{attribute 'qualified_only'}
VAR_GLOBAL
	DigIn AT %I*:ARRAY[1..16]	OF	BOOL;
	DigOut1 AT %Q*:ARRAY[1..4]	OF	BOOL;
	DigOut2 AT %Q*:ARRAY[1..4]	OF	BOOL;
	DigOut3 AT %Q*:ARRAY[1..4]	OF	BOOL;
	DigOut4 AT %Q*:ARRAY[1..4]	OF	BOOL;
	
END_VAR

(* stored: Version 1.1.0.1, ProductVersion 3.1.4024.11
   GVL GVL: Id {606f3125-6c9b-404b-b47a-02777f657aaf} *)
